// TIA Portal V16 export
// export: Created 2024-12-03T15:41:43.5703247Z, ExportSetting WithDefaults, DisplayName Totally Integrated Automation Portal, DisplayVersion V16 Update 6, DisplayName TIA Portal Version Control Interface, DisplayVersion V16 Update 2, DisplayName TIA Portal Openness, DisplayVersion V16 Update 6, DisplayName TIA Portal Teamcenter Gateway, DisplayVersion V16, DisplayName SINAMICS Startdrive Advanced, DisplayVersion V16 Update 5, DisplayName SINAMICS Startdrive G130, G150, S120, S150, SINAMICS MV, S210, DisplayVersion V16 Update 5, DisplayName SINAMICS Startdrive G110M, G120, G120C, G120D, G120P, G115D, DisplayVersion V16 Update 5, DisplayName STEP 7 Professional, DisplayVersion V16 Update 6, DisplayName STEP 7 Safety, DisplayVersion V16, DisplayName WinCC Advanced / Unified PC, DisplayVersion V16 Update 6
FUNCTION_BLOCK "Single_click_FB"   // FB114, SCL
{ S7_Optimized_Access := 'TRUE' }
VERSION : 0.1
// stored: AutoNumber true, IsIECCheckEnabled false, IsRetainMemResEnabled false, MemoryReserve 100, SetENOAutomatically false, UDAEnableTagReadback false
   VAR_INPUT
      I_Signal : "SmartBooldt";
   END_VAR
   VAR_OUTPUT
      O_SignalClick : Bool;
   END_VAR
   VAR
      iddle : TON_TIME;
      buttonPressed : TON_TIME;
      noButtonPress { S7_SetPoint := 'True'} : TON_TIME;
      stepnumber { S7_SetPoint := 'True'} : Int;
   END_VAR
BEGIN
   REGION STEP 10 CAPTURE CLICK

       IF #stepnumber = 0 THEN
           #stepnumber := 10;
       END_IF;

       IF #iddle.Q AND #I_Signal.LE AND #stepnumber = 10 THEN
           #stepnumber := 20;
       END_IF;

   END_REGION

   REGION STEP 20 CHECK BUTTON NOT PRESSED TO LONG

       #buttonPressed(IN := #I_Signal.State,
                      PT := t#1s);

       IF #buttonPressed.Q AND #stepnumber = 20 THEN
           #stepnumber := 10;
       END_IF;

   END_REGION

   REGION STEP 20 BUTTON RELEASED

       IF #I_Signal.FE AND #stepnumber = 20 AND NOT #buttonPressed.Q THEN
           #stepnumber := 30;
       END_IF;

   END_REGION

   REGION STEP 30 CHECK THERE IS NO CLICK X TIME AFTER

       #noButtonPress(IN := #stepnumber = 30,
                      PT := t#800ms);

       IF #stepnumber = 30 AND #I_Signal.LE THEN
           #stepnumber := 10;
       END_IF;

       #O_SignalClick := FALSE;
       IF #noButtonPress.Q THEN
           #O_SignalClick := true;
           #stepnumber := 10;
       END_IF;

   END_REGION

   REGION CHECK IF BUTTON WAS IDDLE

           #iddle(IN := NOT #I_Signal.State,
                  PT := t#1500ms);

   END_REGION
END_FUNCTION_BLOCK
